FUNCTION subVec3 : vec3d
VAR_IN_OUT CONSTANT
	i_vec1 :Vec3d;
	i_vec2 :Vec3d;
END_VAR
VAR
	i: INT ;
END_VAR

FOR i:=1 TO 3 DO 
	subVec3[i]:=i_vec1[i]-i_vec2[i];
END_FOR

END_FUNCTION

(* stored: Version 1.1.0.1, ProductVersion 3.1.4024.12
   POU subVec3: Id {cfdf1d78-21de-4b04-926a-9bbfa26c1fa6}, SpecialFunc None *)
